// TIA Portal V20 export
TYPE "LKinCtrl_typeFrame"
   STRUCT
      x : LReal;   // Translation in x
      y : LReal;   // Translation in y
      z : LReal;   // Translation in z
      "a" : LReal;   // Rotation around z axis
      "b" : LReal;   // Rotation around y axis
      c : LReal;   // Roataion around x axis
   END_STRUCT;
END_TYPE
